{attribute 'enable_dynamic_creation'}
FUNCTION_BLOCK OpcUaDAWriteRequestItem EXTENDS OpcUaDARequestItem
VAR_STAT
	//! <summary>Class name shared by all instances of this function block.</summary>
	_ClassName : STRING := __POUNAME();
END_VAR
VAR
	_Write : Tc3_PLCopen_OpcUa.UA_Write;
END_VAR

{attribute 'monitoring' := 'call'}
PROPERTY ClassName : REFERENCE TO STRING
GET
ClassName REF= _ClassName;
END_GET
END_PROPERTY

//!<param name="namespaceUri">empty string if index used</param>

//!<param name="namespaceIndex">zero if namespace uri used</param>

METHOD Initialize
VAR_INPUT
	namespaceUri : STRING(Tc2_System.MAX_STRING_LENGTH); 
	namespaceIndex : UINT; 
	identifierType : Tc3_PLCopen_OpcUa.E_UAIdentifierType;
	identifier : STRING(Tc2_System.MAX_STRING_LENGTH);
	nodeAdditionalInfo : Tc3_PLCopen_OpcUa.ST_UANodeAdditionalInfo;
	sourceVariable : __SYSTEM.AnyType;
	operationTimeout : TIME := Tc2_System.DEFAULT_ADS_TIMEOUT;
END_VAR
IF namespaceUri <> '' THEN
	_NamespaceUri := namespaceUri;
	_NodeId.nNamespaceIndex := 0;
	_NamespaceIndexValid := FALSE;
ELSE
	_NamespaceUri := '';
	_NodeId.nNamespaceIndex := namespaceIndex;
	_NamespaceIndexValid := TRUE;
END_IF

_NodeId.eIdentifierType := identifierType;
_NodeId.sIdentifier := identifier;

_Write.stNodeAddInfo := nodeAdditionalInfo;
_Write.pVariable := sourceVariable.pValue;
_Write.cbData := TO_UDINT(sourceVariable.diSize);

_GetNodeHandle.Timeout := operationTimeout;
_Write.Timeout := operationTimeout;
_ReleaseNodeHandle.Timeout := operationTimeout;
END_METHOD

METHOD PerformAction : OPC_UA_ACTION_EXECUTION_STATE
VAR_OUTPUT
	exception : Exception;
END_VAR
PerformAction := OPC_UA_ACTION_EXECUTION_STATE.DONE;
	
_Write(Execute := TRUE, ConnectionHdl := _ConnectionHandle, NodeHdl := _GetNodeHandle.NodeHdl);
		
IF _Write.Error THEN
	ExceptionHelper.Throw(
		_Write.ErrorID,
		WString.Concat5("UA_Write error ", TO_WSTRING(_Write.ErrorID), " (Node identifier = '", TO_WSTRING(_NodeId.sIdentifier), "')"),
		__POUNAME(),
		ClassName,
		CurrentNamespace.Name,
		__POSITION(
	)
	);
	PerformAction := OPC_UA_ACTION_EXECUTION_STATE.ERROR;				
	AdsLogger.LogMessage(
		LOGGING_LEVEL.INFORMATION,
		WString.Concat3(
			"---OpcUaRequest performAction error: ",
			"UA_Write error ",
			TO_WSTRING(_Write.ErrorID)
		)
	);
ELSIF _Write.Busy THEN
	PerformAction := OPC_UA_ACTION_EXECUTION_STATE.BUSY;			
END_IF
END_METHOD

METHOD ResetAction
_Write(Execute := FALSE);
END_METHOD

END_FUNCTION_BLOCK

(* stored: Version 1.1.0.1
   POU OpcUaDAWriteRequestItem: Id {e3e8d40a-215f-401d-8ee6-38214d283f4c}, SpecialFunc None
   Property ClassName: Id {40b4228c-0576-46c6-89f7-8bb5492db6f1}
   Get Get: Id {1ed2d809-810b-438a-9368-803451eb5e7b}
   Method Initialize: Id {1fbc5f53-e6fe-4be8-acbe-20048cbe21dd}
   Method PerformAction: Id {eb3df5c7-c55f-4c68-95dc-373f94543e7d}
   Method ResetAction: Id {f5d72c6d-a517-4822-b81c-08f52e85c8de} *)
